// Mitsubishi GX Works2 project: 시퀀스 타이머 회로 1 (간략화)   PLC: Q03UDV

PROGRAM MAIN
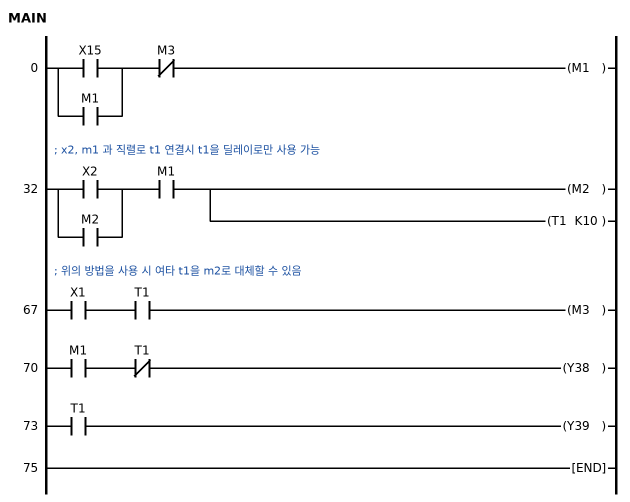
0     LD      X15
      OR      M1
      ANI     M3
      OUT     M1
; x2, m1 과 직렬로 t1 연결시 t1을 딜레이로만 사용 가능
32    LD      X2
      OR      M2
      AND     M1
      OUT     M2
      OUT     T1 K10
; 위의 방법을 사용 시 여타 t1을 m2로 대체할 수 있음
67    LD      X1
      AND     T1
      OUT     M3
70    LD      M1
      ANI     T1
      OUT     Y38
73    LD      T1
      OUT     Y39
75    END
END_PROGRAM
